TYPE AX5000_S_0079 :
STRUCT
	Rotational_position_resolution:UDINT;
END_STRUCT
END_TYPE

(* stored: Version 1.1.0.1, ProductVersion 3.1.4024.3
   DUT AX5000_S_0079: Id {ffabbf13-7998-4fbd-9800-ea464fa2649c} *)
